# EPICS substitutions: viocs/si_ps/si_psApp/Db/sfa0.substitutions
file "db/individual.db" {
    pattern { family, pos, num }
        { "SFA0", "01M1", "" }
        { "SFA0", "01M2", "" }
        { "SFA0", "05M1", "" }
        { "SFA0", "05M2", "" }
        { "SFA0", "09M1", "" }
        { "SFA0", "09M2", "" }
        { "SFA0", "13M1", "" }
        { "SFA0", "13M2", "" }
        { "SFA0", "17M1", "" }
        { "SFA0", "17M2", "" }
}
